SUBAPPLICATION Uebung_012a (* Numeric Value Input und Speichern *)
  (* Standard: 61499-2 *)
  (* Version 1.0, 2023-10-23, franz *)
  FBS
    CbVtStatus : CbVtStatus;
  END_FBS
  SUBAPPS
    Uebung_012a_sub : Uebung_012a_sub(KEY := KEY_I1_STORE, u16ObjId := InputNumber_I1);
  END_SUBAPPS
  EVENT_CONNECTIONS
    CbVtStatus.IND TO Uebung_012a_sub.REQ;
  END_CONNECTIONS
END_SUBAPPLICATION
